PROGRAM P_Demo_FB_DMXGetStatusMessages
VAR
    fbGetStatusMsgs   : FB_DMXGetStatusMessages;      // 读设备状态消息
    stDmxCmdBuffer    : ST_DMXCommandBuffer;          // 与通讯 FB 共用
    wTargetManufId    : WORD := 16#4241;              // 目标灯具厂商 ID
    dwTargetDeviceId  : DWORD := 16#12131415;         // 目标灯具设备 ID
    byTargetPort      : BYTE := 0;                    // 根设备通道 0
    eWantStatusType   : E_DMXStatusType := eDMXStatusTypeError;  // 只读错误级
    bDoRead           : BOOL := FALSE;                // 在线给一次上升沿触发
    bBusy             : BOOL;
    bError            : BOOL;
    udiErrId          : UDINT;
    arrStatusMsgs     : ARRAY [0..24] OF ST_DMXStatusMessage;  // 状态消息数组
END_VAR

// ============================================================
// Tc2_DMX.FB_DMXGetStatusMessages 演示程序
// ============================================================
// 场景：灯光系统集中故障诊断：周期轮询每盏灯的错误级状态消息，汇总到中控 HMI 报警列表。
// 价值：把分散在各灯具的状态/错误信息统一收进 PLC，集中式故障监控，不必逐台本地查看。
// 验证：设 eWantStatusType:=eDMXStatusTypeError，给 bDoRead 一次上升沿 -> bBusy 短暂 TRUE -> 回 FALSE 后 arrStatusMsgs[0..] 含设备当前错误消息（无错误时为空）。
// 验证步骤：
//   1. 右键 PLC 项目下 POUs 文件夹 → Add → Existing Item → 选本 .TcPOU 文件
//   2. 引用 Tc2_DMX；同项目里放一个 FB_EL6851CommunicationEx 实例并共用 stDmxCmdBuffer（非 CycleMode）
//   3. 编译 → 登录 → 运行；按上方『验证』行在线给上升沿观察
// ============================================================

fbGetStatusMsgs(
    bStart                     := bDoRead,
    wDestinationManufacturerId := wTargetManufId,
    dwDestinationDeviceId      := dwTargetDeviceId,
    byPortId                   := byTargetPort,
    eStatusType                := eWantStatusType,
    dwOptions                  := 0,
    stCommandBuffer            := stDmxCmdBuffer,
    bBusy                      => bBusy,
    bError                     => bError,
    udiErrorId                 => udiErrId,
    arrStatusMessages          => arrStatusMsgs
);

END_PROGRAM

(* stored: Version 1.1.0.1, ProductVersion 3.1.4024.5
   POU P_Demo_FB_DMXGetStatusMessages: Id {6076ce96-3c1c-5699-b2e1-7f11be263e9a}, SpecialFunc None *)
